TYPE U64 : ULINT; END_TYPE

(* stored: Version 1.1.0.1
   DUT U64: Id {454be7c8-3b9d-01d1-33d5-5d7a2ecf166a} *)
